FUNCTION Convert_DT_TO_STRING : Hresult
VAR_INPUT
	in : DT;
	out : REFERENCE TO STRING;
END_VAR
VAR
	converted : STRING;
END_VAR
VAR CONSTANT
	INCOMPATIBLE : HRESULT := 16#9811070E;
END_VAR

converted := DT_TO_STRING(in);

IF (STRING_TO_DT(converted) <> in) THEN
	Convert_DT_TO_STRING := INCOMPATIBLE;
	RETURN;
END_IF

out := converted;

END_FUNCTION

(* stored: Version 1.1.0.1, ProductVersion 3.1.4024.12
   POU Convert_DT_TO_STRING: Id {d0c53969-cfda-4fde-ae31-59206521ebf7}, SpecialFunc None *)
